PROGRAM handlesoftEXCEPTION
VAR
	zero : LREAL := 0.000000001;	// Account for floating point representation
END_VAR

(* Handle firmware/HMI exceptions by stopping GVL.appRUN *)

// Handle HMI invalid ranges
IF GVL.chargeTIMEmanual < -1 OR GVL.circuitcapcitanceuF <= zero OR GVL.targetPSUVOLT <= zero OR GVL.psuVOLTrating <= zero OR GVL.psuPOWERpeak <= zero OR GVL.chargeTIMEmanual >60 THEN
	GVL.ctrlsysFAULT := TRUE;
	GVL.softexceptionFAULT:= TRUE;
END_IF

END_PROGRAM

(* stored: Version 1.1.0.1, ProductVersion 3.1.4024.11
   POU handlesoftEXCEPTION: Id {da90aa83-dcd5-40ee-8da1-bce65c6b6d05}, SpecialFunc None *)
